// TIA Portal project "PLC控制V20" (V17)

(* hardware
DEVICE "S7-1500/ET200MP station_1"  S7-1500 station
   slot 0: "导轨_0"  Rack  6ES7 590-1***0-0AA0
   slot 1: "PLC_1"  CPU 1512C-1 PN  6ES7 512-1CK01-0AB0  V2.9
      slot 3: "CPU 显示_1"  6ES7591-1AA00-0AA0
      slot 32768: "PROFINET 接口_1"  X1
         slot 32769: "端口_1"  X1 P1
         slot 32770: "端口_2"  X1 P2
      slot 34817: "Virtual CP interface port_1"  Virtual CP interface port  Virtual CP interface port
*)

// ===== PLC "PLC_1"  CPU 1512C-1 PN =====

VAR_GLOBAL   // PLC tag table "默认变量表"
   "模拟量输入2.1" AT %IB6 : Byte;
   "模拟量输入2.2" AT %IB7 : Byte;
   "启动循环" AT %M0.2 : Bool;
END_VAR

VAR_GLOBAL   // PLC tag table "变量表_1"
   "输出转速的模拟量" AT %QW0 : Int;
   "控制电机正转" AT %M0.0 : Bool;
   "控制电机反转" AT %M0.1 : Bool;
   "电机正转" AT %Q4.1 : Bool;
   "电机反转" AT %Q4.2 : Bool;
   "模拟量输入1.1" AT %IB2 : Byte;
   "模拟量输入1.2" AT %IB3 : Byte;
   "输出电机转速" AT %MD0 : Real;
END_VAR

DATA_BLOCK "PID"   // DB1
{ S7_Optimized_Access := 'FALSE' }
VERSION : 0.1
   VAR
      初始输入的频率 : Int;
      输出转速 : Real;
      输出风速 : Real;
      输出风速_1 : Real;
      累计误差 : Real;
      "风速误差(k)" : Real;
      "风速误差(k-1)" : Real;
      误差差值 : Real;
      控制电机正转 : Bool;
      Kp : Int;
      Kd : Int;
      Ki : Int;
      指定风速 : Real;
      启动循环 : Bool;
      基准Kp : DInt;
      控制电机反转 : Bool;
      区间 : DInt;
      "Kp(i)" : DInt;
      "1" : Real;
      "2" : Real;
   END_VAR
BEGIN
END_DATA_BLOCK

DATA_BLOCK "测量"   // DB2
{ S7_Optimized_Access := 'FALSE' }
VERSION : 0.1
   VAR
      测量启动1 : Bool;
      状态1 : Int;
      状态2 : Int;
      测量电机转速 : Int;
      测量风速 : Real;
      基准Kp : Int;
      状态3 : Int;
      状态4 : Int;
      区间比例 : Real;
      测量启动2 : Bool;
      转速最大量程 : DInt;
      指定风速对应的转速 : DInt;
      指定风速对应的转速_1 : DInt;
      测量启动3 : Bool;
      测量启动4 : Bool;
   END_VAR
BEGIN
END_DATA_BLOCK

FUNCTION "控制电机转速" : Void   // FC1, LAD
{ S7_Optimized_Access := 'TRUE' }
VERSION : 0.1
   VAR_TEMP
      转速比例1 : Real;
      转速比例2 : Real;
      模拟量输入1 : Word;
      输出转速 : Real;
   END_VAR
BEGIN

REGION Network 1: 控制电机转速
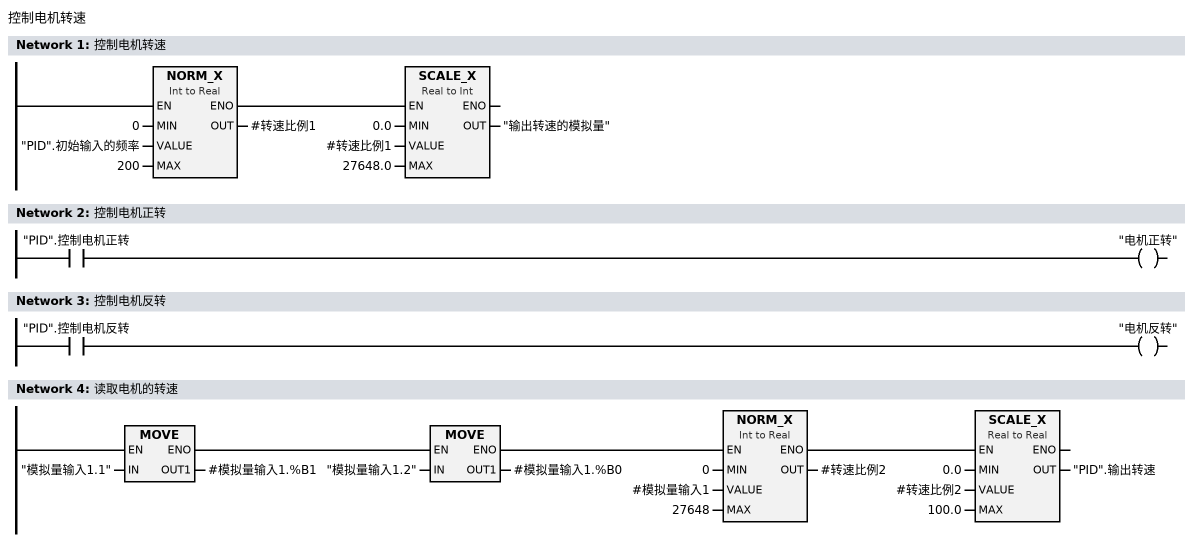
   RUNG wire#powerrail
      { S7_Templates := "[SrcType := Int, DestType := Real]" } Normalize(min := 0, value := "PID".初始输入的频率, max := 200, out => #转速比例1)
      { S7_Templates := "[SrcType := Real, DestType := Int]" } Scale(min := 0.0, value := #转速比例1, max := 27648.0, out => "输出转速的模拟量")
   END_RUNG
   // the same network as SCL:
   #转速比例1 := NORM_X(MIN := 0, VALUE := "PID".初始输入的频率, MAX := 200);
   "输出转速的模拟量" := SCALE_X(MIN := 0.0, VALUE := #转速比例1, MAX := 27648.0);
END_REGION

REGION Network 2: 控制电机正转
   RUNG wire#powerrail
      Contact( "PID".控制电机正转 )
      Coil( "电机正转" )
   END_RUNG
   // the same network as SCL:
   "电机正转" := "PID".控制电机正转;
END_REGION

REGION Network 3: 控制电机反转
   RUNG wire#powerrail
      Contact( "PID".控制电机反转 )
      Coil( "电机反转" )
   END_RUNG
   // the same network as SCL:
   "电机反转" := "PID".控制电机反转;
END_REGION

REGION Network 4: 读取电机的转速
   RUNG wire#powerrail
      Move(in := "模拟量输入1.1", out1 => #模拟量输入1.%B1)
      Move(in := "模拟量输入1.2", out1 => #模拟量输入1.%B0)
      { S7_Templates := "[SrcType := Int, DestType := Real]" } Normalize(min := 0, value := #模拟量输入1, max := 27648, out => #转速比例2)
      { S7_Templates := "[SrcType := Real, DestType := Real]" } Scale(min := 0.0, value := #转速比例2, max := 100.0, out => "PID".输出转速)
   END_RUNG
   // the same network as SCL:
   #模拟量输入1.%B1 := "模拟量输入1.1";
   #模拟量输入1.%B0 := "模拟量输入1.2";
   #转速比例2 := NORM_X(MIN := 0, VALUE := #模拟量输入1, MAX := 27648);
   "PID".输出转速 := SCALE_X(MIN := 0.0, VALUE := #转速比例2, MAX := 100.0);
END_REGION
END_FUNCTION

FUNCTION "风速" : Void   // FC2, LAD
{ S7_Optimized_Access := 'TRUE' }
VERSION : 0.1
   VAR_TEMP
      模拟量输入2 : Word;
      转速比例3 : Real;
   END_VAR
BEGIN

REGION Network 1
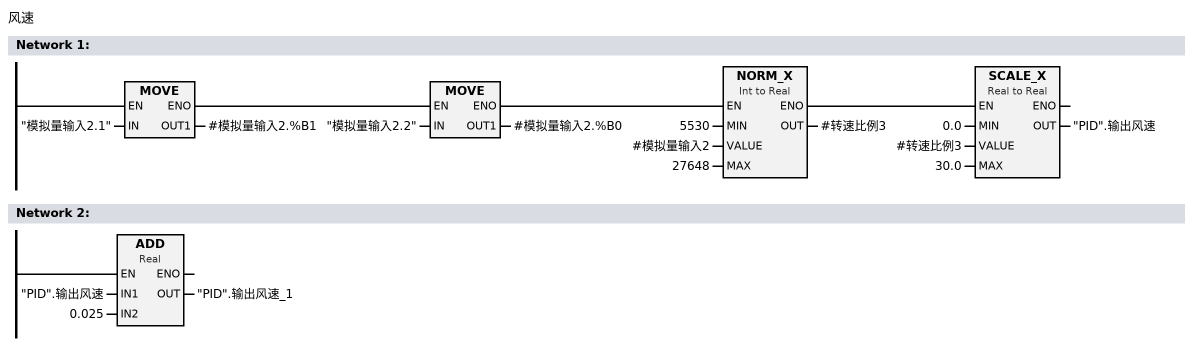
   RUNG wire#powerrail
      Move(in := "模拟量输入2.1", out1 => #模拟量输入2.%B1)
      Move(in := "模拟量输入2.2", out1 => #模拟量输入2.%B0)
      { S7_Templates := "[SrcType := Int, DestType := Real]" } Normalize(min := 5530, value := #模拟量输入2, max := 27648, out => #转速比例3)
      { S7_Templates := "[SrcType := Real, DestType := Real]" } Scale(min := 0.0, value := #转速比例3, max := 30.0, out => "PID".输出风速)
   END_RUNG
   // the same network as SCL:
   #模拟量输入2.%B1 := "模拟量输入2.1";
   #模拟量输入2.%B0 := "模拟量输入2.2";
   #转速比例3 := NORM_X(MIN := 5530, VALUE := #模拟量输入2, MAX := 27648);
   "PID".输出风速 := SCALE_X(MIN := 0.0, VALUE := #转速比例3, MAX := 30.0);
END_REGION

REGION Network 2
   RUNG wire#powerrail
      { S7_Templates := "SrcType := Real" } Add(in1 := "PID".输出风速, in2 := 0.025, out => "PID".输出风速_1)
   END_RUNG
   // the same network as SCL:
   "PID".输出风速_1 := "PID".输出风速 + 0.025;
END_REGION
END_FUNCTION

FUNCTION "控制电机转速SCL_PID" : Void   // FC3, SCL
{ S7_Optimized_Access := 'TRUE' }
VERSION : 0.1
BEGIN
   "PID".Kp := "PID"."Kp(i)";
   IF "PID".启动循环 THEN

       "PID"."风速误差(k)" := "PID".指定风速 - "PID".输出风速_1;
       "PID".误差差值 := "PID"."风速误差(k)"- "PID"."风速误差(k-1)";
       "PID".初始输入的频率 := "PID".初始输入的频率 +("PID"."风速误差(k)" * "PID".Kp) + ("PID".误差差值 * "PID".Kd) + ("PID".累计误差 * "PID".Ki);
       "PID"."风速误差(k-1)" := "PID"."风速误差(k)";
       "PID".累计误差:="PID".累计误差 + "PID"."风速误差(k)";
       ;
   END_IF;
END_FUNCTION

FUNCTION "控制电机转速SCL_P" : Void   // FC5, SCL
{ S7_Optimized_Access := 'TRUE' }
VERSION : 0.1
   VAR_TEMP
      风速误差 : Real;
      Kp : Real;
      指定风速 : Real;
   END_VAR
BEGIN
   #Kp := 10;
   #指定风速 := 3.0;
   IF "启动循环" THEN

       IF "PID".输出风速<#指定风速 THEN
           #风速误差 := #指定风速 - "PID".输出风速_1;
           "PID".初始输入的频率 := "PID".初始输入的频率 + (#风速误差 * #Kp);
           ;
       END_IF;
       IF "PID".输出风速 > #指定风速 THEN
           #风速误差 := "PID".输出风速_1 - #指定风速;
           "PID".初始输入的频率 := "PID".初始输入的频率 - (#风速误差 * #Kp);
           ;
       END_IF;
       ;
   END_IF;
END_FUNCTION

ORGANIZATION_BLOCK "Main"   // OB1, LAD, ProgramCycle
TITLE = "Main Program Sweep (Cycle)"
{ S7_Optimized_Access := 'TRUE' }
VERSION : 0.1
   VAR_INPUT
      Initial_Call : Bool;   // Initial call of this OB
      Remanence : Bool;   // =True, if remanent data are available
   END_VAR
BEGIN

REGION Network 1
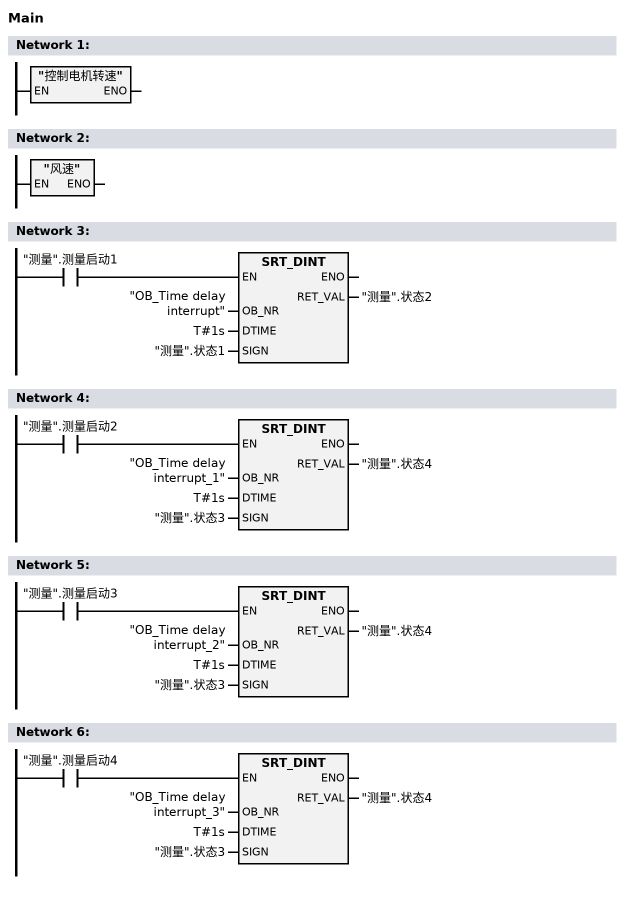
   RUNG wire#powerrail
      "控制电机转速"()
   END_RUNG
   // the same network as SCL:
   "控制电机转速"();
END_REGION

REGION Network 2
   RUNG wire#powerrail
      "风速"()
   END_RUNG
   // the same network as SCL:
   "风速"();
END_REGION

REGION Network 3
   IF "测量".测量启动1 THEN
       "测量".状态2 := SRT_DINT(OB_NR := "OB_Time delay interrupt", DTIME := T#1s, SIGN := "测量".状态1);
   END_IF;
END_REGION

REGION Network 4
   IF "测量".测量启动2 THEN
       "测量".状态4 := SRT_DINT(OB_NR := "OB_Time delay interrupt_1", DTIME := T#1s, SIGN := "测量".状态3);
   END_IF;
END_REGION

REGION Network 5
   IF "测量".测量启动3 THEN
       "测量".状态4 := SRT_DINT(OB_NR := "OB_Time delay interrupt_2", DTIME := T#1s, SIGN := "测量".状态3);
   END_IF;
END_REGION

REGION Network 6
   IF "测量".测量启动4 THEN
       "测量".状态4 := SRT_DINT(OB_NR := "OB_Time delay interrupt_3", DTIME := T#1s, SIGN := "测量".状态3);
   END_IF;
END_REGION
END_ORGANIZATION_BLOCK

ORGANIZATION_BLOCK "Time delay interrupt"   // OB20, SCL, TimeDelayInterrupt
{ S7_Optimized_Access := 'TRUE' }
VERSION : 0.1
   VAR_INPUT
      Sign : Word;   // Identifier input (SIGN) passed to triggering call of SRT_DINT
   END_VAR
   VAR_TEMP
      最大转速 : Int;
   END_VAR
BEGIN
   "PID".初始输入的频率 := "测量".转速最大量程 * "测量".区间比例;
   "测量".测量电机转速 := "测量".转速最大量程 * "测量".区间比例;
END_ORGANIZATION_BLOCK

ORGANIZATION_BLOCK "Time delay interrupt_1"   // OB21, SCL, TimeDelayInterrupt
{ S7_Optimized_Access := 'TRUE' }
VERSION : 0.1
   VAR_INPUT
      Sign : Word;   // Identifier input (SIGN) passed to triggering call of SRT_DINT
   END_VAR
BEGIN
   "测量".测量风速 := "PID".输出风速_1;
   "测量".基准Kp:= "测量".测量电机转速/ "测量".测量风速;
END_ORGANIZATION_BLOCK

ORGANIZATION_BLOCK "Time delay interrupt_2"   // OB22, SCL, TimeDelayInterrupt
{ S7_Optimized_Access := 'TRUE' }
VERSION : 0.1
   VAR_INPUT
      Sign : Word;   // Identifier input (SIGN) passed to triggering call of SRT_DINT
   END_VAR
BEGIN
   "PID".初始输入的频率 := "测量".指定风速对应的转速;
END_ORGANIZATION_BLOCK

ORGANIZATION_BLOCK "Time delay interrupt_3"   // OB23, SCL, TimeDelayInterrupt
{ S7_Optimized_Access := 'TRUE' }
VERSION : 0.1
   VAR_INPUT
      Sign : Word;   // Identifier input (SIGN) passed to triggering call of SRT_DINT
   END_VAR
BEGIN
   "PID".初始输入的频率 := "测量".指定风速对应的转速_1;
END_ORGANIZATION_BLOCK

ORGANIZATION_BLOCK "Cyclic interrupt"   // OB30, LAD, CyclicInterrupt
{ S7_Optimized_Access := 'TRUE' }
VERSION : 0.1
   VAR_INPUT
      Initial_Call : Bool;   // Initial call of this OB
      Event_Count : Int;   // Events discarded
   END_VAR
BEGIN

REGION Network 1
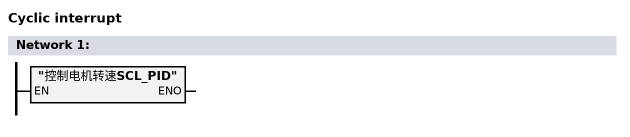
   RUNG wire#powerrail
      "控制电机转速SCL_PID"()
   END_RUNG
   // the same network as SCL:
   "控制电机转速SCL_PID"();
END_REGION
END_ORGANIZATION_BLOCK